TYPE ST_TestData :
STRUCT
    bFlag : BOOL;
    nCount : INT := 0;
END_STRUCT
END_TYPE

(* stored: Version 1.1.0.1
   DUT ST_TestData: Id {55555555-5555-5555-5555-555555555502} *)
